PROGRAM MAIN
VAR
	fb_velocity : FB_MoveVelocity;
	//fb_test : FB_AxisBase;
END_VAR

fb_velocity(axis_ref := GVL.axis_a);
//fb_test(axis_ref := GVL.axis_a);

END_PROGRAM

(* stored: Version 1.1.0.1, ProductVersion 3.1.4024.12
   POU MAIN: Id {d9502940-2ecc-4413-8856-226e3cb8fc00}, SpecialFunc None *)
